// Mitsubishi GX Works2 project: PLC_자기유지회로   PLC: Q03UD

PROGRAM MAIN
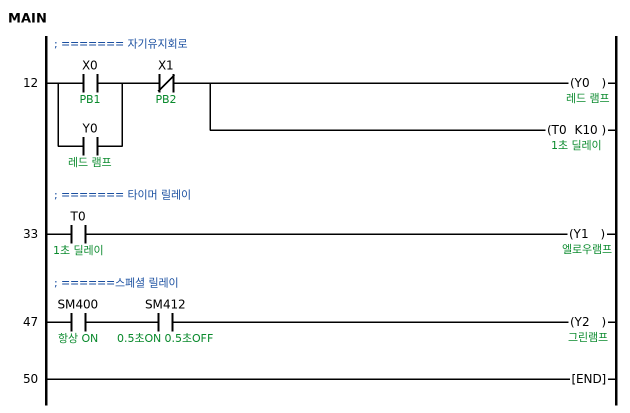
; ======= 자기유지회로
12    LD      X0  ; PB1
      OR      Y0  ; 레드 램프
      ANI     X1  ; PB2
      OUT     Y0  ; 레드 램프
      OUT     T0 K10  ; 1초 딜레이
; ======= 타이머 릴레이
33    LD      T0  ; 1초 딜레이
      OUT     Y1  ; 엘로우램프
; ======스페셜 릴레이
47    LD      SM400  ; 항상 ON
      AND     SM412  ; 0.5초ON 0.5초OFF
      OUT     Y2  ; 그린램프
50    END
END_PROGRAM

PROGRAM TL
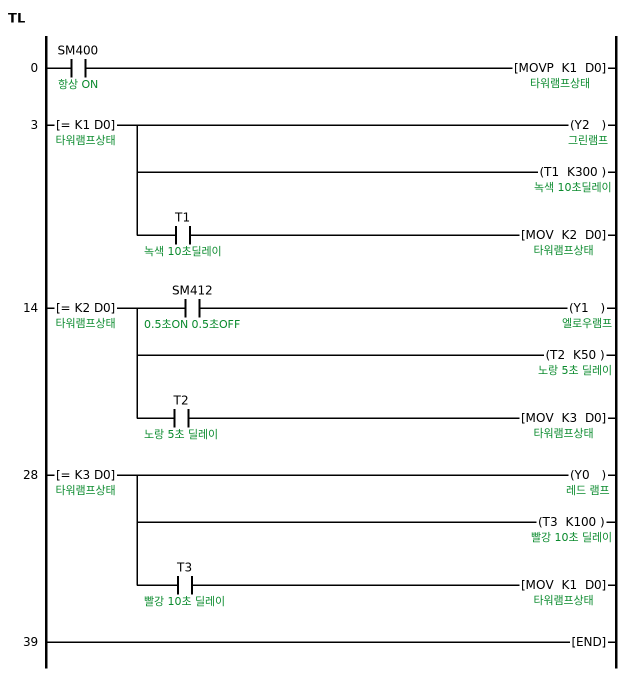
0     LD      SM400  ; 항상 ON
      MOVP    K1 D0  ; 타워램프상태
3     LD=     K1 D0  ; 타워램프상태
      OUT     Y2  ; 그린램프
      OUT     T1 K300  ; 녹색 10초딜레이
      AND     T1  ; 녹색 10초딜레이
      MOV     K2 D0
14    LD=     K2 D0  ; 타워램프상태
      MPS
      AND     SM412  ; 0.5초ON 0.5초OFF
      OUT     Y1  ; 엘로우램프
      MPP
      OUT     T2 K50  ; 노랑 5초 딜레이
      AND     T2  ; 노랑 5초 딜레이
      MOV     K3 D0
28    LD=     K3 D0  ; 타워램프상태
      OUT     Y0  ; 레드 램프
      OUT     T3 K100  ; 빨강 10초 딜레이
      AND     T3  ; 빨강 10초 딜레이
      MOV     K1 D0
39    END
END_PROGRAM

PROGRAM Ex01
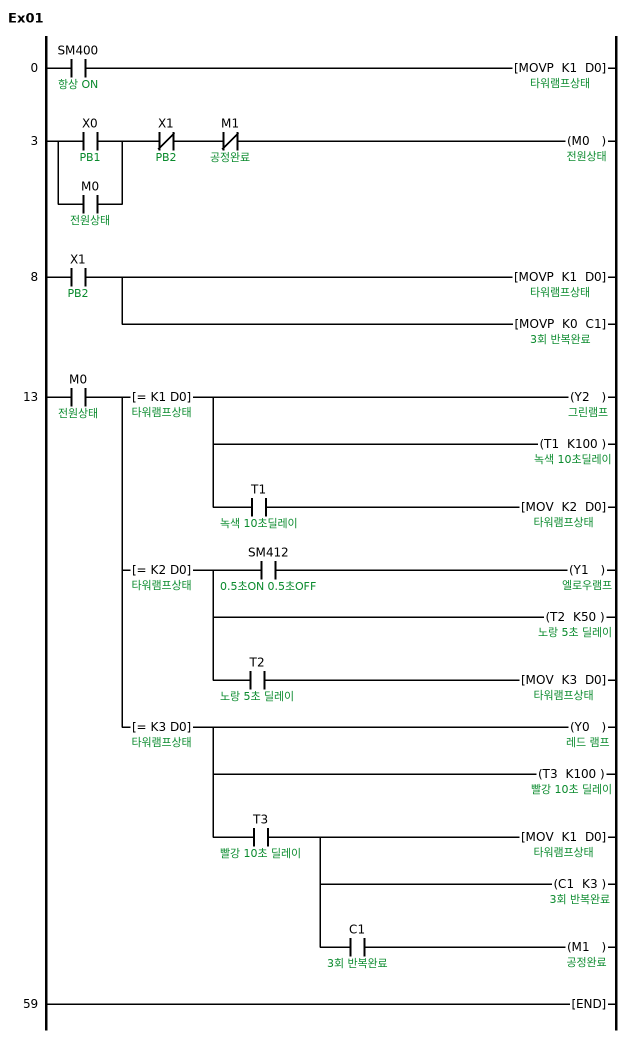
0     LD      SM400  ; 항상 ON
      MOVP    K1 D0  ; 타워램프상태
3     LD      X0  ; PB1
      OR      M0  ; 전원상태
      ANI     X1  ; PB2
      ANI     M1  ; 공정완료
      OUT     M0  ; 전원상태
8     LD      X1  ; PB2
      MOVP    K1 D0
      MOVP    K0 C1  ; 3회 반복완료
13    LD      M0  ; 전원상태
      MPS
      AND=    K1 D0  ; 타워램프상태
      OUT     Y2  ; 그린램프
      OUT     T1 K100  ; 녹색 10초딜레이
      AND     T1  ; 녹색 10초딜레이
      MOV     K2 D0
      MRD
      AND=    K2 D0  ; 타워램프상태
      MPS
      AND     SM412  ; 0.5초ON 0.5초OFF
      OUT     Y1  ; 엘로우램프
      MPP
      OUT     T2 K50  ; 노랑 5초 딜레이
      AND     T2  ; 노랑 5초 딜레이
      MOV     K3 D0
      MPP
      AND=    K3 D0  ; 타워램프상태
      OUT     Y0  ; 레드 램프
      OUT     T3 K100  ; 빨강 10초 딜레이
      AND     T3  ; 빨강 10초 딜레이
      MOV     K1 D0
      OUT     C1 K3  ; 3회 반복완료
      AND     C1  ; 3회 반복완료
      OUT     M1  ; 공정완료
59    END
END_PROGRAM

PROGRAM Counter
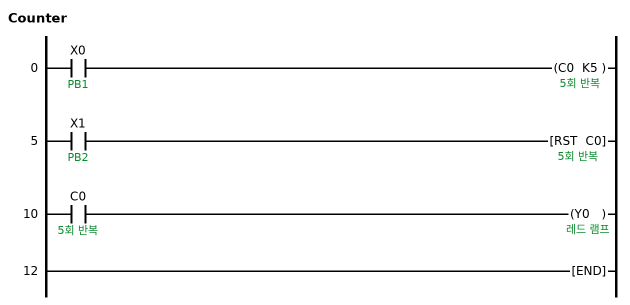
0     LD      X0  ; PB1
      OUT     C0 K5  ; 5회 반복
5     LD      X1  ; PB2
      RST     C0  ; 5회 반복
10    LD      C0  ; 5회 반복
      OUT     Y0  ; 레드 램프
12    END
END_PROGRAM
